// TIA Portal V19 export
FUNCTION_BLOCK "TYPIC_C501_IF_KLH"   // FB63, FBD
TITLE = TYPIC_C501_IF_KLH: Handbediende klep
{ S7_Optimized_Access := 'TRUE' }
AUTHOR : OCOTECH
FAMILY : Typical
NAME : C501.704
// Logisch Object Besturing: C501.704
// 
// De interne functie handbediende klep verzorgt de bewaking van één van volgende componenten:
//  een handbediende klep
//  een leegzetvoorziening
//  een beo/ontluchtingsvoorziening
// stored: MemoryReserve 10, SetENOAutomatically false
   VAR_INPUT
      EXT_HW { ExternalAccessible := 'False'; ExternalVisible := 'False'; ExternalWritable := 'False'} : Bool;   // Sturings hardware (PLC) bewaking (1 = OK)
      IN_OPEN { ExternalAccessible := 'False'; ExternalVisible := 'False'; ExternalWritable := 'False'} : Bool;   // Handbediende klep is open
      IN_TOE { ExternalAccessible := 'False'; ExternalVisible := 'False'; ExternalWritable := 'False'} : Bool;   // Handbediende klep is toe
      CFG_OPEN { ExternalAccessible := 'False'; ExternalVisible := 'False'; ExternalWritable := 'False'} : Bool;   // Handbediende klep heeft een toestandsmelding Open
      CFG_TOE { ExternalAccessible := 'False'; ExternalVisible := 'False'; ExternalWritable := 'False'} : Bool;   // Handbediende klep heeft een toestandsmelding Toe
   END_VAR
   VAR_OUTPUT
      VAR_IF_KLH { ExternalAccessible := 'False'; ExternalVisible := 'False'; ExternalWritable := 'False'} : "C501_VAR_IF_KLH_TYPIC";   // Struct met alle variabelen naar bovenliggende functies
   END_VAR
   VAR
      STO { ExternalWritable := 'False'} : Struct   // Storingen
         A001 : Bool;   // Terugmeldingen Open en Dicht tegelijk
      END_STRUCT;
      VAR { ExternalWritable := 'False'} : Struct   // Variabelen
         STS_OPEN : Bool;   // Handbediende klep is open
         STS_TOE : Bool;   // Handbediende klep is toe
         EXT_HW { ExternalAccessible := 'False'; ExternalVisible := 'False'} : Bool;   // Sturings hardware (PLC) in storing
      END_STRUCT;
   END_VAR
BEGIN

REGION Network 1: START
END_REGION

REGION Network 2: +++ Status +++
   // De status van de handbediende klep (open / dicht) wordt doorgestuurd naar 3B.
END_REGION

REGION Network 3: +++ Storingen +++
   // Alle storingen worden doorgegeven aan 3B.
END_REGION

REGION Network 4: Storing A001: Terugmeldingen Open en Dicht tegelijk
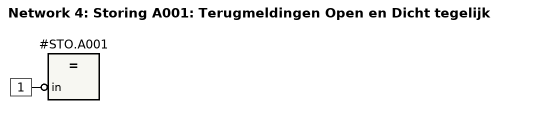
   #STO.A001 := NOT 1;
END_REGION

REGION Network 5 (SCL): EINDE
   // Variabelen van intern scada rakvlak naar outputs copieren
   #VAR_IF_KLH.STS_OPEN := #VAR.STS_OPEN;
   #VAR_IF_KLH.STS_TOE := #VAR.STS_TOE;
   #VAR_IF_KLH.EXT_HW := #VAR.EXT_HW;
   #VAR_IF_KLH.STO := #STO;
END_REGION
END_FUNCTION_BLOCK
